FUNCTION FUN_BuildLogString : String
VAR_INPUT
	fPos : LREAL;
	fVelocity : LREAL;
	fGap : LREAL;
END_VAR
VAR
	sTemp: STRING;
END_VAR

sTemp := 				CONCAT('Pos:' , LREAL_TO_STRING(fPos));
sTemp := CONCAT(sTemp, 	CONCAT(', Velocity:' , LREAL_TO_STRING(fVelocity)));
sTemp := CONCAT(sTemp, 	CONCAT(', Gap:' , LREAL_TO_STRING(fGap)));

FUN_BuildLogString := sTemp;

END_FUNCTION

(* stored: Version 1.1.0.1, ProductVersion 3.1.4024.12
   POU FUN_BuildLogString: Id {672fc2ac-58d1-4618-9b9b-db68825d7425}, SpecialFunc None *)
